FUNCTION IsValidIterator : BOOL
VAR_INPUT
    Iterator : ITcVnIteratorBase;
END_VAR

IsValidIterator := Iterator <> 0;

END_FUNCTION

(* stored: Version 1.1.0.1, ProductVersion 3.1.4024.13
   POU IsValidIterator: Id {fe2c5c3f-8d10-0565-0c59-737e9caa00d2}, SpecialFunc None *)
